// TIA Portal V20 export
// export: Created 2026-04-10T20:43:33Z, ExportSetting WithDefaults
DATA_BLOCK "TP307"   // DB1
{ S7_Optimized_Access := 'TRUE' }
   VAR
      drive1 : Struct
         blocked { S7_SetPoint := 'True'} : "messageConfig_UDT";
         communicationError { S7_SetPoint := 'True'} : "messageConfig_UDT";
      END_STRUCT;
      drive2 : Struct
         blocked { S7_SetPoint := 'True'} : "messageConfig_UDT";
      END_STRUCT;
   END_VAR
BEGIN
   drive1.blocked.moduleId := 10;
   drive1.blocked.elementId := 1;
   drive1.blocked.messageId := 101;
   drive1.communicationError.moduleId := 10;
   drive1.communicationError.elementId := 1;
   drive1.communicationError.messageId := 102;
   drive2.blocked.moduleId := 20;
   drive2.blocked.elementId := 2;
   drive2.blocked.messageId := 201;
END_DATA_BLOCK
